PROGRAM MAIN
VAR
	Pippo	: BOOL;
	Paperino : BOOL;
	Pluto	: BBOL;
END_VAR

Pippo := TRUE;
Paperino := TRUE;

END_PROGRAM

(* stored: Version 1.1.0.1, ProductVersion 3.1.4024.13
   POU MAIN: Id {c2782fdd-b80e-4ae7-a3a3-9440492aedf8}, SpecialFunc None *)
